PROGRAM Std_System_Out
VAR

	Clk50ms:TON;
	ClkOff50ms:TON;
	Clk100ms:TON;
	ClkOff100ms:TON;
	Clk500ms:TON;
	ClkOff500ms:TON;
	ClkOn1s:TON;
	ClkOff1s:TON;

	T50ms_RTRIG: R_TRIG;
	T100ms_RTRIG: R_TRIG;
	T500ms_RTRIG: R_TRIG;
	T1s_RTRIG: R_TRIG;

END_VAR

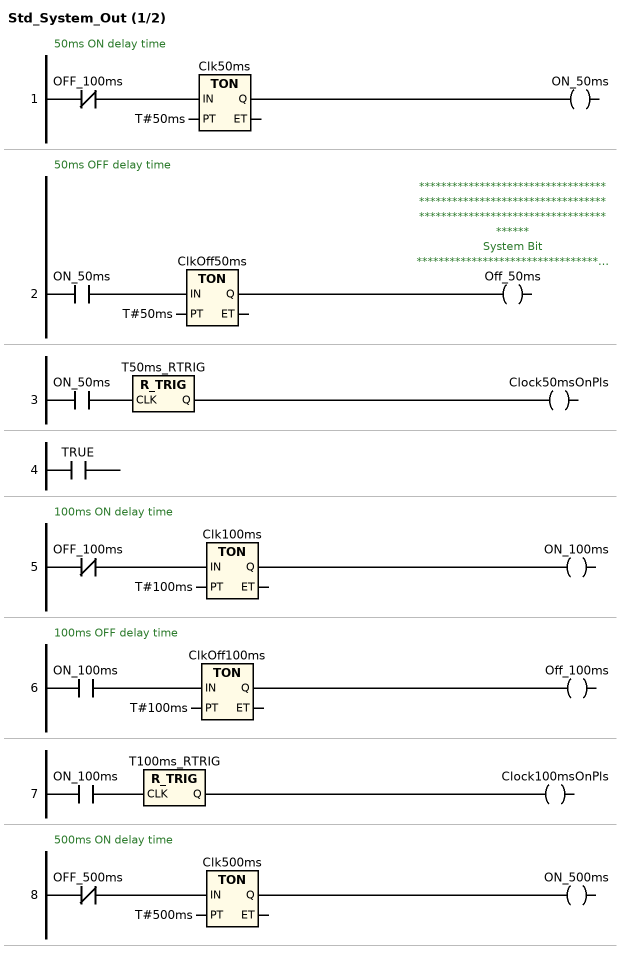
// NETWORK 1
// 50ms ON delay time
Clk50ms(IN := NOT OFF_100ms, PT := T#50ms); // TON
ON_50ms := Clk50ms.Q;

// NETWORK 2
// 50ms OFF delay time
//   Off_50ms: ************************************************************************************************************ System Bit ************************************************************************************************************
ClkOff50ms(IN := ON_50ms, PT := T#50ms); // TON
Off_50ms := ClkOff50ms.Q;

// NETWORK 3
T50ms_RTRIG(CLK := ON_50ms); // R_TRIG
Clock50msOnPls := T50ms_RTRIG.Q;

// NETWORK 4

// NETWORK 5
// 100ms ON delay time
Clk100ms(IN := NOT OFF_100ms, PT := T#100ms); // TON
ON_100ms := Clk100ms.Q;

// NETWORK 6
// 100ms OFF delay time
ClkOff100ms(IN := ON_100ms, PT := T#100ms); // TON
Off_100ms := ClkOff100ms.Q;

// NETWORK 7
T100ms_RTRIG(CLK := ON_100ms); // R_TRIG
Clock100msOnPls := T100ms_RTRIG.Q;

// NETWORK 8
// 500ms ON delay time
Clk500ms(IN := NOT OFF_500ms, PT := T#500ms); // TON
ON_500ms := Clk500ms.Q;

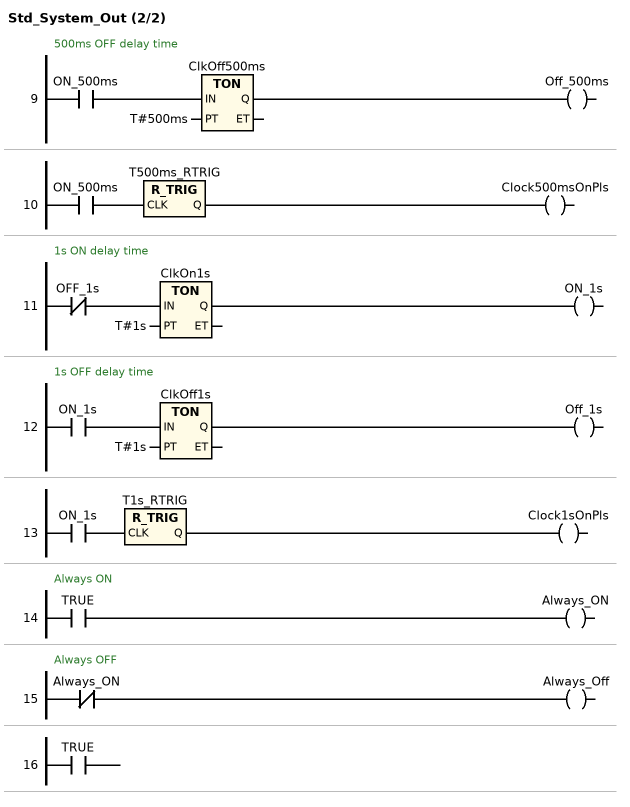
// NETWORK 9
// 500ms OFF delay time
ClkOff500ms(IN := ON_500ms, PT := T#500ms); // TON
Off_500ms := ClkOff500ms.Q;

// NETWORK 10
T500ms_RTRIG(CLK := ON_500ms); // R_TRIG
Clock500msOnPls := T500ms_RTRIG.Q;

// NETWORK 11
// 1s ON delay time
ClkOn1s(IN := NOT OFF_1s, PT := T#1s); // TON
ON_1s := ClkOn1s.Q;

// NETWORK 12
// 1s OFF delay time
ClkOff1s(IN := ON_1s, PT := T#1s); // TON
Off_1s := ClkOff1s.Q;

// NETWORK 13
T1s_RTRIG(CLK := ON_1s); // R_TRIG
Clock1sOnPls := T1s_RTRIG.Q;

// NETWORK 14
// Always ON
Always_ON := TRUE;

// NETWORK 15
// Always OFF
Always_Off := NOT Always_ON;

// NETWORK 16

END_PROGRAM

(* stored: Version 1.1.0.1, ProductVersion 3.1.4018.5
   POU Std_System_Out: Id {cd901e8a-f6e4-413b-ba9b-fe3707c5df81}, SpecialFunc None *)
